FUNCTION_BLOCK FB_LamparaTemporizada_LD
// La lampara se enciende al accionar el pulsador
// La lampara se apaga transcurrido un tiempo encendida
VAR_INPUT
    TiempoEncendido   : TIME := T#2S;
END_VAR
VAR_OUTPUT
    TiempoPendiente   : TIME;
END_VAR
VAR
    Temporizador      : TON;
    Memoria           : RS;
    Lampara   AT %Q*  : BOOL;
    Pulsador  AT %I*  : BOOL;
END_VAR

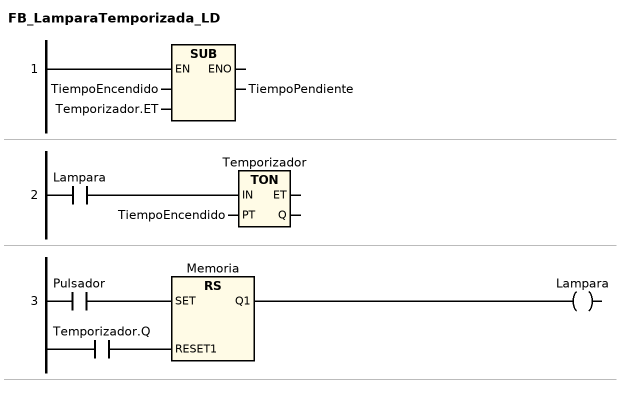
// NETWORK 1
TiempoPendiente := TiempoEncendido - Temporizador.ET;

// NETWORK 2
Temporizador(IN := Lampara, PT := TiempoEncendido); // TON

// NETWORK 3
Memoria(SET := Pulsador, RESET1 := Temporizador.Q); // RS
Lampara := Memoria.Q1;

END_FUNCTION_BLOCK

(* stored: Version 1.1.0.1, ProductVersion 3.1.4024.15
   POU FB_LamparaTemporizada_LD: Id {424061ba-8d78-48c7-b4ae-26f15978acd8}, SpecialFunc None *)
